{attribute 'linkalways'} 
{attribute 'no_explicit_call' := 'This FB is a CLASS and must be accessed using methods or properties'}
{attribute 'enable_dynamic_creation'}
FUNCTION_BLOCK Node_F_VN_ImageAverageStdDevExp EXTENDS VisionNode
VAR
    ipSrcImage : _ITcVnImage;
    aAverage : _TcVnVector4_LREAL;
    aStdDev : _TcVnVector4_LREAL;
    ipMask : _ITcVnImage;
    hrPrev : _HRESULT(S_OK);
	hresult : _HRESULT(S_OK);
END_VAR

METHOD PUBLIC  Clone : I_Node
VAR
	pNode : POINTER TO Node_F_VN_ImageAverageStdDevExp;
END_VAR
pNode := __NEW(Node_F_VN_ImageAverageStdDevExp);
Clone := pNode^;
END_METHOD

METHOD FB_init : BOOL
VAR_INPUT
	bInitRetains : BOOL; // if TRUE, the retain variables are initialized (warm start / cold start)
	bInCopyCode : BOOL;  // if TRUE, the instance afterwards gets moved into the copy code (online change)
END_VAR
AddInput('ipSrcImage', ipSrcImage);
AddInput('ipMask', ipMask);
AddInput('hrPrev', hrPrev);
AddOutput('aAverage', aAverage);
AddOutput('aStdDev', aStdDev);
AddOutput('hresult', hresult);
END_METHOD

METHOD PROTECTED OnExecute
hresult.Value := F_VN_ImageAverageStdDevExp(
	ipSrcImage := ipSrcImage.Value,
    aAverage := aAverage.Value,
    aStdDev := aStdDev.Value,
    ipMask := ipMask.Value,
	hrPrev:= hrPrev.Value);
END_METHOD

METHOD PUBLIC PreExecutionCheck
VAR_INPUT
	Check : I_PreExecutionChecks;
END_VAR
Check.IsTrue(ipSrcImage.IsValid, 'ipSrcImage must contain an image');
Check.IsTrue((ipSrcImage.HasChannelCount(1) OR
              ipSrcImage.HasChannelCount(2) OR
              ipSrcImage.HasChannelCount(3) OR
              ipSrcImage.HasChannelCount(4)), 'ipSrcImage must contain 1, 2, 3 or 4 channels');

Check.IsTrue(ipMask.IsValid, 'ipMask must contain an image');
Check.IsTrue(ipMask.HasChannelCount(1), 'ipMask must have 1 channel');
Check.IsTrue(ipMask.IsPixelDepth(8), 'ipMask must have 8 bit pixel depth');
Check.IsTrue(IsImage1SizeEqualToImage2Size(ipMask.Value, ipSrcImage.Value), 'ipMask must be the same size as ipSrcImage');
END_METHOD

END_FUNCTION_BLOCK

(* stored: Version 1.1.0.1, ProductVersion 3.1.4024.13
   POU Node_F_VN_ImageAverageStdDevExp: Id {1a1de6cd-4a03-0e93-3793-eb1ae644d049}, SpecialFunc None
   Folder Constructor: Id {5c77058d-ff09-0850-3247-018e81afd21d}
   Method Clone: Id {637b0f33-48a9-0f67-31db-028356885323}
   Method FB_init: Id {6a9021c9-47be-0b63-0e2e-0b5f9780c7eb}
   Method OnExecute: Id {c6b45329-d399-0e24-117f-78fab64fe4ac}
   Method PreExecutionCheck: Id {bf92260c-4a6e-056e-0fa2-095a420e0cc9} *)
